(* IEC 61131-3 sources: SRCI/RobotLibrary/Library/POUs/BasicMove/MC_MoveAxesAbsolute, 1 file *)

(* ---- MC_MoveAxesAbsoluteFB.st ---- *)
/// Move all joints to an absolute joint position (Absolute Joint PTP)
FUNCTION_BLOCK MC_MoveAxesAbsoluteFB EXTENDS RobotLibraryBaseExecuteFB
// -------------------------------------------------------------------------
//  SRCI Robot Library
// -------------------------------------------------------------------------
//
//  Object:      MoveAxesAbsoluteFB
//  Author:      Thorsten Brach
//  Date:        2024-06-01
//
//  Description:
//
//
//  Copyright:
//    (C) 2024 Thorsten Brach. All rights reserved
//             Licensed under the LGPL-3.0 license.
//
//  Disclaimer:
//    This project is provided without any guarantee and can be used for
//    private and commercial purposes. Any use is at the user’s
//    own risk and responsibility.
//
// -------------------------------------------------------------------------
VAR_INPUT
  /// Parameter which determines the behavior towards the previously sent and still active or buffered commands
  AbortingMode       : AbortingMode;
  /// Defines the target sequence in which the command will be executed
  SequenceFlag       : SequenceFlag;
  /// command parameter
  ParCmd             : MoveAxesAbsoluteParCmd;
END_VAR

VAR_OUTPUT
  /// Command is transferred and confirmed by the RC
  CommandBuffered    : BOOL;
  /// The command takes control of the motion of the according axis group
  Active             : BOOL;
  /// The command was aborted by another command.
  CommandAborted     : BOOL;
  /// TRUE, while command is interrupted during execution and can be continued
  CommandInterrupted : BOOL;
  /// command results
  OutCmd             : MoveAxesAbsoluteOutCmd;
END_VAR

VAR
  /// internal copy of command parameter
 _parCmd             : MoveAxesAbsoluteParCmd;
  /// command data to send
 _command            : MoveAxesAbsoluteSendData;
  /// response data received
 _response           : MoveAxesAbsoluteRecvData;
END_VAR

  SUPER^(AxesGroup := AxesGroup);

END_FUNCTION_BLOCK

METHOD INTERNAL CheckAddParameter : BOOL
VAR_INPUT
  /// Payload pointer
  PayloadPtr : UDINT;
END_VAR
VAR
  /// Payload as byte array
  Payload    : ARRAY [1..SIZEOF(_command)] OF BYTE;
  /// Null Byte array
  Null       : ARRAY [1..SIZEOF(_command)] OF BYTE;
  /// Data length to compare
  DataLen    : UDINT;
END_VAR

  // Payload pointer must be decreased by one byte, because ADR(Payload) is already one byte !
  PayloadPtr := LIMIT (0, PayloadPtr - 1, SIZEOF(Payload) -1);
  // Convert command struct to payload array
  SysDepMemCpy( pDest := ADR(Payload), pSrc := ADR(_command), DataLen := SIZEOF(_command));
  // Calculate the data length to compare - at least one byte must be compared !
  DataLen := LIMIT(1, SIZEOF(Payload) - PayloadPtr, SIZEOF(Payload));
  // Compare Payload-Array with Null-Byte-Array
  CheckAddParameter := SysDepMemCmp( pData1 := ADR(Payload) + PayloadPtr , pData2 := ADR(Null), DataLen := DataLen) <>  RobotLibraryConstants.OK ;

END_METHOD

METHOD PROTECTED CheckFunctionSupported : BOOL
VAR_IN_OUT
  /// Robot assignment of function
  AxesGroup : AxesGroup;
END_VAR

  CheckFunctionSupported := AxesGroup.State.RobotData.RCSupportedFunctions.MoveAxesAbsolute;

  IF ( NOT CheckFunctionSupported )
  THEN
    // call base implementation for set error and create log entry
    SUPER^.CheckFunctionSupported(AxesGroup := AxesGroup);
  END_IF

END_METHOD

METHOD PROTECTED CheckParameterChanged : BOOL
VAR_IN_OUT
  /// Robot assignment of function
  AxesGroup    : AxesGroup;
END_VAR

  // Check ParCmd Size is > 0, because MemCmp does not work correctly with size = 0
  IF (SIZEOF(ParCmd) = 0) OR (_stepCmd = 0)
  THEN
    RETURN;
  END_IF

  // compare memory
  _parameterChanged := ( SysDepMemCmp(pData1 := ADR(ParCmd), pData2 := ADR(_parCmd), DataLen := SIZEOF(ParCmd)) <> RobotLibraryConstants.OK );

  // check parameter valid ?
  _parameterValid   := CheckParameterValid( AxesGroup := AxesGroup );

  IF ((  _parameterChanged        )  AND
      (  _parameterValid          )) OR
      (  _parameterUpdateInternal )
  THEN
    // reset internal flag for send parameter update
   _parameterUpdateInternal := FALSE;
    // update internal copy of parameters
   _parCmd := ParCmd;
    // inc parameter sequence
   _command.ParSeq := _command.ParSeq + 1;
    // update command data
    CommandData := CreateCommandPayload(AxesGroup := AxesGroup); // ( Access via reference to rCommandFB in ACR )
    // notify active command register
    AxesGroup.Acyclic.ActiveCommandRegister.NotifyParameterChanged := _uniqueID;
  END_IF

END_METHOD

METHOD PROTECTED CheckParameterValid : BOOL
VAR_IN_OUT
  /// Robot assignment of function
  AxesGroup : AxesGroup;
END_VAR
VAR
  /// internal index for loops
 _idx : DINT;
END_VAR

  CheckParameterValid := TRUE;

  // Check AbortingMode valid ?
  IF (( AbortingMode <> AbortingModeEnum.BUFFER ) AND
      ( AbortingMode <> AbortingModeEnum.ABORT  ))
  THEN
    // Parameter not valid
    CheckParameterValid := FALSE;
    // Set error
    ErrorID := RobotLibraryErrorIdEnum.ERR_ABORTINGMODE_INVALID;
    // Create log entry
    CreateLogMessagePara1 ( Timestamp   := AxesGroup.State.SystemTime,
                            MessageType := MessageType.CMD,
                            Severity    := Severity.ERROR,
                            MessageCode := ErrorID,
                            MessageText := 'Invalid Parameter AbortingMode = {1}',
                            Para1       := ABORTING_MODE_TO_STRING(AbortingMode));
    RETURN;
  END_IF

  // Check SequenceFlag valid ?
  IF (( SequenceFlag <> SequenceFlagEnum.PRIMARY_SEQUENCE   ) AND
      ( SequenceFlag <> SequenceFlagEnum.SECONDARY_SEQUENCE ))
  THEN
    // Parameter not valid
    CheckParameterValid := FALSE;
    // Set error
    ErrorID := RobotLibraryErrorIdEnum.ERR_SEQFLAG_NOT_ALLOWED;
    // Create log entry
    CreateLogMessagePara1 ( Timestamp   := AxesGroup.State.SystemTime,
                            MessageType := MessageType.CMD,
                            Severity    := Severity.ERROR,
                            MessageCode := ErrorID,
                            MessageText := 'Invalid Parameter SequenceFlag = {1}',
                            Para1       := SEQUENCE_FLAG_TO_STRING(SequenceFlag));
    RETURN;
  END_IF

  // Check ParCmd.JointPosition.J1 valid ?
  IF ( SysDepIsValidReal(ParCmd.JointPosition.J1) = FALSE )
  THEN
    // Parameter not valid
    CheckParameterValid := FALSE;
    // Set error
    ErrorID := RobotLibraryErrorIdEnum.ERR_INVALID_PAR_CMD;

    // Create log entry
    CreateLogMessagePara1 ( Timestamp   := AxesGroup.State.SystemTime,
                            MessageType := MessageType.CMD,
                            Severity    := Severity.ERROR,
                            MessageCode := ErrorID,
                            MessageText := 'Invalid Parameter ParCmd.JointPosition.J1 = {1}',
                            Para1       := VALID_REAL_TO_STRING(ParCmd.JointPosition.J1));
    RETURN;
  END_IF

  // Check ParCmd.JointPosition.J2 valid ?
  IF ( SysDepIsValidReal(ParCmd.JointPosition.J2) = FALSE )
  THEN
    // Parameter not valid
    CheckParameterValid := FALSE;
    // Set error
    ErrorID := RobotLibraryErrorIdEnum.ERR_INVALID_PAR_CMD;

    // Create log entry
    CreateLogMessagePara1 ( Timestamp   := AxesGroup.State.SystemTime,
                            MessageType := MessageType.CMD,
                            Severity    := Severity.ERROR,
                            MessageCode := ErrorID,
                            MessageText := 'Invalid Parameter ParCmd.JointPosition.J2 = {1}',
                            Para1       := VALID_REAL_TO_STRING(ParCmd.JointPosition.J2));
    RETURN;
  END_IF

  // Check ParCmd.JointPosition.J3 valid ?
  IF ( SysDepIsValidReal(ParCmd.JointPosition.J3) = FALSE )
  THEN
    // Parameter not valid
    CheckParameterValid := FALSE;
    // Set error
    ErrorID := RobotLibraryErrorIdEnum.ERR_INVALID_PAR_CMD;

    // Create log entry
    CreateLogMessagePara1 ( Timestamp   := AxesGroup.State.SystemTime,
                            MessageType := MessageType.CMD,
                            Severity    := Severity.ERROR,
                            MessageCode := ErrorID,
                            MessageText := 'Invalid Parameter ParCmd.JointPosition.J3 = {1}',
                            Para1       := VALID_REAL_TO_STRING(ParCmd.JointPosition.J3));
    RETURN;
  END_IF

  // Check ParCmd.JointPosition.J4 valid ?
  IF ( SysDepIsValidReal(ParCmd.JointPosition.J4) = FALSE )
  THEN
    // Parameter not valid
    CheckParameterValid := FALSE;
    // Set error
    ErrorID := RobotLibraryErrorIdEnum.ERR_INVALID_PAR_CMD;

    // Create log entry
    CreateLogMessagePara1 ( Timestamp   := AxesGroup.State.SystemTime,
                            MessageType := MessageType.CMD,
                            Severity    := Severity.ERROR,
                            MessageCode := ErrorID,
                            MessageText := 'Invalid Parameter ParCmd.JointPosition.J4 = {1}',
                            Para1       := VALID_REAL_TO_STRING(ParCmd.JointPosition.J4));
    RETURN;
  END_IF

  // Check ParCmd.JointPosition.J5 valid ?
  IF ( SysDepIsValidReal(ParCmd.JointPosition.J5) = FALSE )
  THEN
    // Parameter not valid
    CheckParameterValid := FALSE;
    // Set error
    ErrorID := RobotLibraryErrorIdEnum.ERR_INVALID_PAR_CMD;

    // Create log entry
    CreateLogMessagePara1 ( Timestamp   := AxesGroup.State.SystemTime,
                            MessageType := MessageType.CMD,
                            Severity    := Severity.ERROR,
                            MessageCode := ErrorID,
                            MessageText := 'Invalid Parameter ParCmd.JointPosition.J5 = {1}',
                            Para1       := VALID_REAL_TO_STRING(ParCmd.JointPosition.J5));
    RETURN;
  END_IF

  // Check ParCmd.JointPosition.J6 valid ?
  IF ( SysDepIsValidReal(ParCmd.JointPosition.J6) = FALSE )
  THEN
    // Parameter not valid
    CheckParameterValid := FALSE;
    // Set error
    ErrorID := RobotLibraryErrorIdEnum.ERR_INVALID_PAR_CMD;

    // Create log entry
    CreateLogMessagePara1 ( Timestamp   := AxesGroup.State.SystemTime,
                            MessageType := MessageType.CMD,
                            Severity    := Severity.ERROR,
                            MessageCode := ErrorID,
                            MessageText := 'Invalid Parameter ParCmd.JointPosition.J6 = {1}',
                            Para1       := VALID_REAL_TO_STRING(ParCmd.JointPosition.J6));
    RETURN;
  END_IF

  // Check ParCmd.JointPosition.E1 valid ?
  IF ( SysDepIsValidReal(ParCmd.JointPosition.E1) = FALSE )
  THEN
    // Parameter not valid
    CheckParameterValid := FALSE;
    // Set error
    ErrorID := RobotLibraryErrorIdEnum.ERR_INVALID_PAR_CMD;

    // Create log entry
    CreateLogMessagePara1 ( Timestamp   := AxesGroup.State.SystemTime,
                            MessageType := MessageType.CMD,
                            Severity    := Severity.ERROR,
                            MessageCode := ErrorID,
                            MessageText := 'Invalid Parameter ParCmd.JointPosition.E1 = {1}',
                            Para1       := VALID_REAL_TO_STRING(ParCmd.JointPosition.E1));
    RETURN;
  END_IF

  // Check ParCmd.JointPosition.E2 valid ?
  IF ( SysDepIsValidReal(ParCmd.JointPosition.E2) = FALSE )
  THEN
    // Parameter not valid
    CheckParameterValid := FALSE;
    // Set error
    ErrorID := RobotLibraryErrorIdEnum.ERR_INVALID_PAR_CMD;

    // Create log entry
    CreateLogMessagePara1 ( Timestamp   := AxesGroup.State.SystemTime,
                            MessageType := MessageType.CMD,
                            Severity    := Severity.ERROR,
                            MessageCode := ErrorID,
                            MessageText := 'Invalid Parameter ParCmd.JointPosition.E2 = {1}',
                            Para1       := VALID_REAL_TO_STRING(ParCmd.JointPosition.E2));
    RETURN;
  END_IF

  // Check ParCmd.JointPosition.E3 valid ?
  IF ( SysDepIsValidReal(ParCmd.JointPosition.E3) = FALSE )
  THEN
    // Parameter not valid
    CheckParameterValid := FALSE;
    // Set error
    ErrorID := RobotLibraryErrorIdEnum.ERR_INVALID_PAR_CMD;

    // Create log entry
    CreateLogMessagePara1 ( Timestamp   := AxesGroup.State.SystemTime,
                            MessageType := MessageType.CMD,
                            Severity    := Severity.ERROR,
                            MessageCode := ErrorID,
                            MessageText := 'Invalid Parameter ParCmd.JointPosition.E3 = {1}',
                            Para1       := VALID_REAL_TO_STRING(ParCmd.JointPosition.E3));
    RETURN;
  END_IF

  // Check ParCmd.JointPosition.E4 valid ?
  IF ( SysDepIsValidReal(ParCmd.JointPosition.E4) = FALSE )
  THEN
    // Parameter not valid
    CheckParameterValid := FALSE;
    // Set error
    ErrorID := RobotLibraryErrorIdEnum.ERR_INVALID_PAR_CMD;

    // Create log entry
    CreateLogMessagePara1 ( Timestamp   := AxesGroup.State.SystemTime,
                            MessageType := MessageType.CMD,
                            Severity    := Severity.ERROR,
                            MessageCode := ErrorID,
                            MessageText := 'Invalid Parameter ParCmd.JointPosition.E4 = {1}',
                            Para1       := VALID_REAL_TO_STRING(ParCmd.JointPosition.E4));
    RETURN;
  END_IF

  // Check ParCmd.JointPosition.E5 valid ?
  IF ( SysDepIsValidReal(ParCmd.JointPosition.E5) = FALSE )
  THEN
    // Parameter not valid
    CheckParameterValid := FALSE;
    // Set error
    ErrorID := RobotLibraryErrorIdEnum.ERR_INVALID_PAR_CMD;

    // Create log entry
    CreateLogMessagePara1 ( Timestamp   := AxesGroup.State.SystemTime,
                            MessageType := MessageType.CMD,
                            Severity    := Severity.ERROR,
                            MessageCode := ErrorID,
                            MessageText := 'Invalid Parameter ParCmd.JointPosition.E5 = {1}',
                            Para1       := VALID_REAL_TO_STRING(ParCmd.JointPosition.E5));
    RETURN;
  END_IF

  // Check ParCmd.JointPosition.E6 valid ?
  IF ( SysDepIsValidReal(ParCmd.JointPosition.E6) = FALSE )
  THEN
    // Parameter not valid
    CheckParameterValid := FALSE;
    // Set error
    ErrorID := RobotLibraryErrorIdEnum.ERR_INVALID_PAR_CMD;

    // Create log entry
    CreateLogMessagePara1 ( Timestamp   := AxesGroup.State.SystemTime,
                            MessageType := MessageType.CMD,
                            Severity    := Severity.ERROR,
                            MessageCode := ErrorID,
                            MessageText := 'Invalid Parameter ParCmd.JointPosition.E6 = {1}',
                            Para1       := VALID_REAL_TO_STRING(ParCmd.JointPosition.E6));
    RETURN;
  END_IF

  // Check ParCmd.VelocityRate valid ?
  IF  (( SysDepIsValidReal(ParCmd.VelocityRate) = FALSE )  OR
      ((                   ParCmd.VelocityRate  <     0 )  AND
       (                   ParCmd.VelocityRate <>    -1 )) OR
       (                   ParCmd.VelocityRate  >   100 ))
  THEN
    // Parameter not valid
    CheckParameterValid := FALSE;
    // Set error
    ErrorID := RobotLibraryErrorIdEnum.ERR_VELOCITY_INVALID;
    // Create log entry
    CreateLogMessagePara1 ( Timestamp   := AxesGroup.State.SystemTime,
                            MessageType := MessageType.CMD,
                            Severity    := Severity.ERROR,
                            MessageCode := ErrorID,
                            MessageText := 'Invalid Parameter ParCmd.VelocityRate = {1}',
                            Para1       := VALID_REAL_TO_STRING(ParCmd.VelocityRate));
    RETURN;
  END_IF

  // Check ParCmd.AccelerationRate valid ?
  IF  (( SysDepIsValidReal(ParCmd.AccelerationRate) = FALSE )  OR
      ((                   ParCmd.AccelerationRate  <     0 )  AND
       (                   ParCmd.AccelerationRate <>    -1 )) OR
       (                   ParCmd.AccelerationRate  >   100 ))
  THEN
    // Parameter not valid
    CheckParameterValid := FALSE;
    // Set error
    ErrorID := RobotLibraryErrorIdEnum.ERR_ACCELERATION_INVALID;
    // Create log entry
    CreateLogMessagePara1 ( Timestamp   := AxesGroup.State.SystemTime,
                            MessageType := MessageType.CMD,
                            Severity    := Severity.ERROR,
                            MessageCode := ErrorID,
                            MessageText := 'Invalid Parameter ParCmd.AccelerationRate = {1}',
                            Para1       := VALID_REAL_TO_STRING(ParCmd.AccelerationRate));
    RETURN;
  END_IF

  // Check ParCmd.DecelerationRate valid ?
  IF  (( SysDepIsValidReal(ParCmd.DecelerationRate) = FALSE )  OR
      ((                   ParCmd.DecelerationRate  <     0 )  AND
       (                   ParCmd.DecelerationRate <>    -1 )) OR
       (                   ParCmd.DecelerationRate  >   100 ))
  THEN
    // Parameter not valid
    CheckParameterValid := FALSE;
    // Set error
    ErrorID := RobotLibraryErrorIdEnum.ERR_DECELERATION_INVALID;
    // Create log entry
    CreateLogMessagePara1 ( Timestamp   := AxesGroup.State.SystemTime,
                            MessageType := MessageType.CMD,
                            Severity    := Severity.ERROR,
                            MessageCode := ErrorID,
                            MessageText := 'Invalid Parameter ParCmd.DecelerationRate = {1}',
                            Para1       := VALID_REAL_TO_STRING(ParCmd.DecelerationRate));
    RETURN;
  END_IF

  // Check ParCmd.JerkRate valid ?
  IF  (( SysDepIsValidReal(ParCmd.JerkRate) = FALSE )  OR
      ((                   ParCmd.JerkRate  <     0 )  AND
       (                   ParCmd.JerkRate <>    -1 )) OR
       (                   ParCmd.JerkRate  >   100 ))
  THEN
    // Parameter not valid
    CheckParameterValid := FALSE;
    // Set error
    ErrorID := RobotLibraryErrorIdEnum.ERR_JERK_INVALID;
    // Create log entry
    CreateLogMessagePara1 ( Timestamp   := AxesGroup.State.SystemTime,
                            MessageType := MessageType.CMD,
                            Severity    := Severity.ERROR,
                            MessageCode := ErrorID,
                            MessageText := 'Invalid Parameter ParCmd.JerkRate = {1}',
                            Para1       := VALID_REAL_TO_STRING(ParCmd.JerkRate));
    RETURN;
  END_IF

  // Check ParCmd.ToolNo valid ?
  IF (( ParCmd.ToolNo <   0                                                ) OR
      ( ParCmd.ToolNo > 254                                                ) OR
      ( ParCmd.ToolNo > AxesGroup.State.ConfigurationData.HighestToolIndex ) OR
      ( ParCmd.ToolNo > RobotLibraryParameter.TOOL_MAX -1                  ))
  THEN
    // Parameter not valid
    CheckParameterValid := FALSE;

    // Check ToolNo available on RC ?
    IF ( ParCmd.ToolNo > AxesGroup.State.ConfigurationData.HighestToolIndex )
    THEN
      ErrorID := RobotLibraryErrorIdEnum.ERR_TOOLNO_UNAVAILABLE;
    ELSE
      ErrorID := RobotLibraryErrorIdEnum.ERR_TOOLNO_RANGE;
  	END_IF

    // Create log entry
    CreateLogMessagePara1 ( Timestamp   := AxesGroup.State.SystemTime,
                            MessageType := MessageType.CMD,
                            Severity    := Severity.ERROR,
                            MessageCode := ErrorID,
                            MessageText := 'Invalid Parameter ParCmd.ToolNo = {1}',
                            Para1       := USINT_TO_STRING(ParCmd.ToolNo));
    RETURN;
  END_IF

  // Check ParCmd.BlendingMode valid ?
  IF (( ParCmd.BlendingMode <> BlendingMode.EXACT_STOP           ) AND
      ( ParCmd.BlendingMode <> BlendingMode.DEFINED_VELOCITY     ) AND
      ( ParCmd.BlendingMode <> BlendingMode.CORNER_DISTANCE      ) AND
      ( ParCmd.BlendingMode <> BlendingMode.MAX_CORNER_DEVIATION ) AND
      ( ParCmd.BlendingMode <> BlendingMode.CORNER_DISTANCE_2R   ) AND
      ( ParCmd.BlendingMode <> BlendingMode.RAMP_OVERLAP         ) AND
      ( ParCmd.BlendingMode <> BlendingMode.CORNER_DISTANCE_1R   ))
  THEN
    // Parameter not valid
    CheckParameterValid := FALSE;
    // Set error
    ErrorID := RobotLibraryErrorIdEnum.ERR_INVALID_PAR_CMD;
    // Create log entry
    CreateLogMessagePara1 ( Timestamp   := AxesGroup.State.SystemTime,
                            MessageType := MessageType.CMD,
                            Severity    := Severity.ERROR,
                            MessageCode := ErrorID,
                            MessageText := 'Invalid Parameter ParCmd.BlendingMode = {1}',
                            Para1       := BLENDING_MODE_TO_STRING(ParCmd.BlendingMode));
    RETURN;
  END_IF

  FOR _idx := 0 TO 1
  DO
    // Check ParCmd.BlendingParameter valid ?
    IF  ( SysDepIsValidReal(ParCmd.BlendingParameter[_idx]) = FALSE )
    THEN
      // Parameter not valid
      CheckParameterValid := FALSE;
      // Set error
      ErrorID := RobotLibraryErrorIdEnum.ERR_JERK_INVALID;
      // Create log entry
      CreateLogMessagePara2 ( Timestamp   := AxesGroup.State.SystemTime,
                              MessageType := MessageType.CMD,
                              Severity    := Severity.ERROR,
                              MessageCode := ErrorID,
                              MessageText := 'Invalid Parameter ParCmd.BlendingParameter[{2}] = {1}',
                              Para1       := VALID_REAL_TO_STRING(ParCmd.JerkRate),
                              Para2       := DINT_TO_STRING(_idx));
      EXIT;
      RETURN;
    END_IF
  END_FOR

  // Check ParCmd.MoveTime valid ?
  IF  ( ParCmd.MoveTime < T#0S )
  THEN
    // Parameter not valid
    CheckParameterValid := FALSE;
    // Set error
    ErrorID := RobotLibraryErrorIdEnum.ERR_INVALID_PAR_CMD;
    // Create log entry
    CreateLogMessagePara1 ( Timestamp   := AxesGroup.State.SystemTime,
                            MessageType := MessageType.CMD,
                            Severity    := Severity.ERROR,
                            MessageCode := ErrorID,
                            MessageText := 'Invalid Parameter ParCmd.MoveTime = {1}',
                            Para1       := TIME_TO_STRING(ParCmd.MoveTime));
    RETURN;
  END_IF

  // Check ParCmd.Manipulation
  // -> no plausibility check for boolean

  FOR _idx := 0 TO 3
  DO
    // Check ParCmd.EmitterID valid ?
    IF  (( ParCmd.EmitterID[_idx] < -127 ) OR
         ( ParCmd.EmitterID[_idx] >  127 ))
    THEN
      // Parameter not valid
      CheckParameterValid := FALSE;
      // Set error
      ErrorID := RobotLibraryErrorIdEnum.ERR_INVALID_PAR_CMD;
      // Create log entry
      CreateLogMessagePara2 ( Timestamp   := AxesGroup.State.SystemTime,
                              MessageType := MessageType.CMD,
                              Severity    := Severity.ERROR,
                              MessageCode := ErrorID,
                              MessageText := 'Invalid Parameter ParCmd.EmitterID[{2}] = {1}',
                              Para1       := SINT_TO_STRING(ParCmd.EmitterID[_idx]),
                              Para2       := DINT_TO_STRING(_idx));
      EXIT;
      RETURN;
    END_IF
  END_FOR

END_METHOD

METHOD INTERNAL CreateCommandPayload : RobotLibraryCommandDataFB
VAR_IN_OUT
  /// Robot assignment of function
  AxesGroup : AxesGroup;
END_VAR
VAR
  /// internal index for loops
 _idx          : DINT;
  /// Parameter count
 _parameterCnt : DINT;
END_VAR
// Table 6-261: Sent CMD payload (PLC to RC) of "MoveAxesAbsolute
// --------------------------
// Header
// --------------------------
// --------------------------
// Datablock
// --------------------------
// Byte 00 : UINT  - Type HB
// Byte 01 :       - Type LB
// Byte 02 : USINT - Reserve | ExecutionMode
// Byte 03 : USINT - ParSeq  | Priority
// --------------------------
// Datablock
// --------------------------
// Byte 04 : SINT       - EmitterID[0]
// Byte 05 : SINT       - EmitterID[1]
// Byte 06 : SINT       - EmitterID[2]
// Byte 07 : SINT       - EmitterID[3]
// Byte 08 : SINT       - ListenerID
// Byte 09 : BYTE       - Reserved
// Byte 10 : UINT       - VelocityRate HW HB
// Byte 11 :            - VelocityRate HW LB
// Byte 12 : UINT       - AccelerationRate HW HB
// Byte 13 :            - AccelerationRate HW LB
// Byte 14 : UINT       - DecelerationRate HW HB
// Byte 15 :            - DecelerationRate HW LB
// Byte 16 : UINT       - JerkRate HW HB
// Byte 17 :            - JerkRate HW LB
// Byte 18 : USINT      - ToolNo
// Byte 19 : USINT      - BlendingMode
// Byte 20 : REAL       - BlendingParameter[0] HW HB
// Byte 21 :            - BlendingParameter[0] HW LB
// Byte 22 :            - BlendingParameter[0] LW HB
// Byte 23 :            - BlendingParameter[0] LW LB
// Byte 24 : REAL       - BlendingParameter[1] HW HB
// Byte 25 :            - BlendingParameter[1] HW LB
// Byte 26 :            - BlendingParameter[1] LW HB
// Byte 27 :            - BlendingParameter[1] LW LB
// Byte 28 : REAL       - JointPosition.J1 HW HB
// Byte 29 :            - JointPosition.J1 HW LB
// Byte 30 :            - JointPosition.J1 LW HB
// Byte 31 :            - JointPosition.J1 LW LB
// Byte 32 : REAL       - JointPosition.J2 HW HB
// Byte 33 :            - JointPosition.J2 HW LB
// Byte 34 :            - JointPosition.J2 LW HB
// Byte 35 :            - JointPosition.J2 LW LB
// Byte 36 : REAL       - JointPosition.J3 HW HB
// Byte 37 :            - JointPosition.J3 HW LB
// Byte 38 :            - JointPosition.J3 LW HB
// Byte 39 :            - JointPosition.J3 LW LB
// Byte 40 : REAL       - JointPosition.J4 HW HB
// Byte 41 :            - JointPosition.J4 HW LB
// Byte 42 :            - JointPosition.J4 LW HB
// Byte 43 :            - JointPosition.J4 LW LB
// Byte 44 : REAL       - JointPosition.J5 HW HB
// Byte 45 :            - JointPosition.J5 HW LB
// Byte 46 :            - JointPosition.J5 LW HB
// Byte 47 :            - JointPosition.J5 LW LB
// Byte 48 : REAL       - JointPosition.J6 HW HB
// Byte 49 :            - JointPosition.J6 HW LB
// Byte 50 :            - JointPosition.J6 LW HB
// Byte 51 :            - JointPosition.J6 LW LB
// Byte 52 : REAL       - JointPosition.E1 HW HB
// Byte 53 :            - JointPosition.E1 HW LB
// Byte 54 :            - JointPosition.E1 LW HB
// Byte 55 :            - JointPosition.E1 LW LB
// Byte 56 : BOOL       - Manipulation
// Byte 57 : BYTE       - Reserve
// Byte 58 : UINT       - Time HW HB
// Byte 59 :            - Time HW LB
// Byte 60 : REAL       - JointPosition.E2 HW HB
// Byte 61 :            - JointPosition.E2 HW LB
// Byte 62 :            - JointPosition.E2 LW HB
// Byte 63 :            - JointPosition.E2 LW LB
// Byte 64 : REAL       - JointPosition.E3 HW HB
// Byte 65 :            - JointPosition.E3 HW LB
// Byte 66 :            - JointPosition.E3 LW HB
// Byte 67 :            - JointPosition.E3 LW LB
// Byte 68 : REAL       - JointPosition.E4 HW HB
// Byte 69 :            - JointPosition.E4 HW LB
// Byte 70 :            - JointPosition.E4 LW HB
// Byte 71 :            - JointPosition.E4 LW LB
// Byte 72 : REAL       - JointPosition.E5 HW HB
// Byte 73 :            - JointPosition.E5 HW LB
// Byte 74 :            - JointPosition.E5 LW HB
// Byte 75 :            - JointPosition.E5 LW LB
// Byte 76 : REAL       - JointPosition.E6 HW HB
// Byte 77 :            - JointPosition.E6 HW LB
// Byte 78 :            - JointPosition.E6 LW HB
// Byte 79 :            - JointPosition.E6 LW LB

  // set command parameter
  _command.CmdTyp            :=  CmdType.MoveAxesAbsolute;
  _command.ExecMode          :=  ExecMode;
  _command.ParSeq            := _command.ParSeq;
  _command.Priority          :=  Priority;
  _command.EmitterID[0]      := _parCmd.EmitterID[0];
  _command.EmitterID[1]      := _parCmd.EmitterID[1];
  _command.EmitterID[2]      := _parCmd.EmitterID[2];
  _command.EmitterID[3]      := _parCmd.EmitterID[3];
  _command.ListenerID        := 0;
  _command.Reserve           := 0;

  _command.VelocityRate      := REAL_TO_PERCENT_UINT(_parCmd.VelocityRate     , IsOptional := FALSE);
  _command.AccelerationRate  := REAL_TO_PERCENT_UINT(_parCmd.AccelerationRate , IsOptional := FALSE);
  _command.JerkRate          := REAL_TO_PERCENT_UINT(_parCmd.JerkRate         , IsOptional := TRUE );
  _command.DecelerationRate  := REAL_TO_PERCENT_UINT(_parCmd.DecelerationRate , IsOptional := TRUE );

  _command.ToolNo            := _parCmd.ToolNo;
  _command.BlendingMode      := _parCmd.BlendingMode;
  _command.BlendingParameter := _parCmd.BlendingParameter;
  _command.JointPosition     := _parCmd.JointPosition;
  _command.Manipulation      := _parCmd.Manipulation;
  _command.MoveTime          := TIME_TO_UINT(_parCmd.MoveTime);

  // copy command data to header
  _cmdHeader := _command;
  // call base implementation to copy header to payload buffer
  CreateCommandPayload := SUPER^.CreateCommandPayload(AxesGroup := AxesGroup);

  FOR _idx := 0 TO 3
  DO
    // Check parameter must be added ?
    IF ( CheckAddParameter(CreateCommandPayload.PayloadPtr))
    THEN
      // add command.EmitterID[x]
      CreateCommandPayload.AddSint(_command.EmitterID[_idx]);
      // inc parameter counter
     _parameterCnt := _parameterCnt + 1;
    END_IF
  END_FOR

  // Check parameter must be added ?
  IF ( CheckAddParameter(CreateCommandPayload.PayloadPtr))
  THEN
    // add command.ListenerID
    CreateCommandPayload.AddSint(_command.ListenerID);
    // inc parameter counter
   _parameterCnt := _parameterCnt + 1;
  END_IF

  // Check parameter must be added ?
  IF ( CheckAddParameter(CreateCommandPayload.PayloadPtr))
  THEN
    // add command.Reserve
    CreateCommandPayload.AddSint(_command.Reserve);
    // inc parameter counter
   _parameterCnt := _parameterCnt + 1;
  END_IF

  // Check parameter must be added ?
  IF ( CheckAddParameter(CreateCommandPayload.PayloadPtr))
  THEN
    // add command.VelocityRate
    CreateCommandPayload.AddUint(_command.VelocityRate);
    // inc parameter counter
   _parameterCnt := _parameterCnt + 1;
  END_IF

  // Check parameter must be added ?
  IF ( CheckAddParameter(CreateCommandPayload.PayloadPtr))
  THEN
    // add command.AccelerationRate
    CreateCommandPayload.AddUint(_command.AccelerationRate);
    // inc parameter counter
   _parameterCnt := _parameterCnt + 1;
  END_IF

  // Check parameter must be added ?
  IF ( CheckAddParameter(CreateCommandPayload.PayloadPtr))
  THEN
    // add command.DecelerationRate
    CreateCommandPayload.AddUint(_command.DecelerationRate);
    // inc parameter counter
   _parameterCnt := _parameterCnt + 1;
  END_IF

  // Check parameter must be added ?
  IF ( CheckAddParameter(CreateCommandPayload.PayloadPtr))
  THEN
    // add command.JerkRate
    CreateCommandPayload.AddUint(_command.JerkRate);
    // inc parameter counter
   _parameterCnt := _parameterCnt + 1;
  END_IF

  // Check parameter must be added ?
  IF ( CheckAddParameter(CreateCommandPayload.PayloadPtr))
  THEN
    // add command.ToolNo
    CreateCommandPayload.AddUsint(_command.ToolNo);
    // inc parameter counter
   _parameterCnt := _parameterCnt + 1;
  END_IF

  // Check parameter must be added ?
  IF ( CheckAddParameter(CreateCommandPayload.PayloadPtr))
  THEN
    // add command.BlendingMode
    CreateCommandPayload.AddUsint(_command.BlendingMode);
    // inc parameter counter
   _parameterCnt := _parameterCnt + 1;
  END_IF

  // Check parameter must be added ?
  IF ( CheckAddParameter(CreateCommandPayload.PayloadPtr))
  THEN
    // add command.BlendingParameter[0]
    CreateCommandPayload.AddReal(_command.BlendingParameter[0]);
    // inc parameter counter
   _parameterCnt := _parameterCnt + 1;
  END_IF

  // Check parameter must be added ?
  IF ( CheckAddParameter(CreateCommandPayload.PayloadPtr))
  THEN
    // add command.BlendingParameter[1]
    CreateCommandPayload.AddReal(_command.BlendingParameter[1]);
    // inc parameter counter
   _parameterCnt := _parameterCnt + 1;
  END_IF

  // Check parameter must be added ?
  IF ( CheckAddParameter(CreateCommandPayload.PayloadPtr))
  THEN
    // add command.JointPosition.J1
    CreateCommandPayload.AddReal(_command.JointPosition.J1);
    // inc parameter counter
   _parameterCnt := _parameterCnt + 1;
  END_IF

  // Check parameter must be added ?
  IF ( CheckAddParameter(CreateCommandPayload.PayloadPtr))
  THEN
    // add command.JointPosition.J2
    CreateCommandPayload.AddReal(_command.JointPosition.J2);
    // inc parameter counter
   _parameterCnt := _parameterCnt + 1;
  END_IF

  // Check parameter must be added ?
  IF ( CheckAddParameter(CreateCommandPayload.PayloadPtr))
  THEN
    // add command.JointPosition.J3
    CreateCommandPayload.AddReal(_command.JointPosition.J3);
    // inc parameter counter
   _parameterCnt := _parameterCnt + 1;
  END_IF

  // Check parameter must be added ?
  IF ( CheckAddParameter(CreateCommandPayload.PayloadPtr))
  THEN
    // add command.JointPosition.J4
    CreateCommandPayload.AddReal(_command.JointPosition.J4);
    // inc parameter counter
   _parameterCnt := _parameterCnt + 1;
  END_IF

  // Check parameter must be added ?
  IF ( CheckAddParameter(CreateCommandPayload.PayloadPtr))
  THEN
    // add command.JointPosition.J5
    CreateCommandPayload.AddReal(_command.JointPosition.J5);
    // inc parameter counter
   _parameterCnt := _parameterCnt + 1;
  END_IF

  // Check parameter must be added ?
  IF ( CheckAddParameter(CreateCommandPayload.PayloadPtr))
  THEN
    // add command.JointPosition.J6
    CreateCommandPayload.AddReal(_command.JointPosition.J6);
    // inc parameter counter
   _parameterCnt := _parameterCnt + 1;
  END_IF

  // Check parameter must be added ?
  IF ( CheckAddParameter(CreateCommandPayload.PayloadPtr))
  THEN
    // add command.JointPosition.E1
    CreateCommandPayload.AddReal(_command.JointPosition.E1);
    // inc parameter counter
   _parameterCnt := _parameterCnt + 1;
  END_IF

  // Check parameter must be added ?
  IF ( CheckAddParameter(CreateCommandPayload.PayloadPtr))
  THEN
    // add command.Manipulation
    CreateCommandPayload.AddBool(_command.Manipulation);
    // inc parameter counter
   _parameterCnt := _parameterCnt + 1;
  END_IF

  // Check parameter must be added ?
  IF ( CheckAddParameter(CreateCommandPayload.PayloadPtr))
  THEN
    // add command.Reserve
    CreateCommandPayload.AddByte(_command.Reserve2);
    // inc parameter counter
   _parameterCnt := _parameterCnt + 1;
  END_IF

  // Check parameter must be added ?
  IF ( CheckAddParameter(CreateCommandPayload.PayloadPtr))
  THEN
    // add command.MoveTime
    CreateCommandPayload.AddUint(_command.MoveTime);
    // inc parameter counter
   _parameterCnt := _parameterCnt + 1;
  END_IF

  // Check parameter must be added ?
  IF ( CheckAddParameter(CreateCommandPayload.PayloadPtr))
  THEN
    // add command.JointPosition.E2
    CreateCommandPayload.AddReal(_command.JointPosition.E2);
    // inc parameter counter
   _parameterCnt := _parameterCnt + 1;
  END_IF

  // Check parameter must be added ?
  IF ( CheckAddParameter(CreateCommandPayload.PayloadPtr))
  THEN
    // add command.JointPosition.E3
    CreateCommandPayload.AddReal(_command.JointPosition.E3);
    // inc parameter counter
   _parameterCnt := _parameterCnt + 1;
  END_IF

  // Check parameter must be added ?
  IF ( CheckAddParameter(CreateCommandPayload.PayloadPtr))
  THEN
    // add command.JointPosition.E4
    CreateCommandPayload.AddReal(_command.JointPosition.E4);
    // inc parameter counter
   _parameterCnt := _parameterCnt + 1;
  END_IF

  // Check parameter must be added ?
  IF ( CheckAddParameter(CreateCommandPayload.PayloadPtr))
  THEN
    // add command.JointPosition.E5
    CreateCommandPayload.AddReal(_command.JointPosition.E5);
    // inc parameter counter
   _parameterCnt := _parameterCnt + 1;
  END_IF

  // Check parameter must be added ?
  IF ( CheckAddParameter(CreateCommandPayload.PayloadPtr))
  THEN
    // add command.JointPosition.E6
    CreateCommandPayload.AddReal(_command.JointPosition.E6);
    // inc parameter counter
   _parameterCnt := _parameterCnt + 1;
  END_IF

  // create logging
  CreateCommandPayloadLog(AxesGroup := AxesGroup, ParameterCnt := _parameterCnt);

END_METHOD

METHOD INTERNAL CreateCommandPayloadLog
VAR_IN_OUT
  /// Robot assignment of function
  AxesGroup : AxesGroup;
END_VAR
VAR_INPUT
  /// Parameter count
  ParameterCnt : DINT;
END_VAR
VAR
  /// internal index for loops
 _idx : DINT;
END_VAR

  // Create log entry for Parameter start
  CreateLogMessagePara1 ( Timestamp   := AxesGroup.State.SystemTime,
                          MessageType := MessageType.CMD,
                          Severity    := Severity.DEBUG,
                          MessageCode := 0,
                          MessageText := 'Create command payload with the {1} parameter(s) :',
                          Para1       := DINT_TO_STRING(ParameterCnt));

  // Create log entry for EmitterID[x]
  FOR _idx := 0 TO 3
  DO
    // Return if no parameter is remaining...
    IF ( ParameterCnt = 0 ) THEN RETURN; END_IF
    // dec remaining parameter(s)
    ParameterCnt := ParameterCnt - 1;
    // Create log entry for Command.EmitterID
    CreateLogMessagePara2 ( Timestamp   := AxesGroup.State.SystemTime,
                            MessageType := MessageType.CMD,
                            Severity    := Severity.DEBUG,
                            MessageCode := 0,
                            MessageText := 'Command.EmitterID[{2}] = {1}',
                            Para1       :=  SINT_TO_STRING(_command.EmitterID[_idx]),
                            Para2       :=  DINT_TO_STRING(_idx));
  END_FOR

  // Return if no parameter is remaining...
  IF ( ParameterCnt = 0 ) THEN RETURN; END_IF
  // dec remaining parameter(s)
  ParameterCnt := ParameterCnt - 1;
  // Create log entry for ListenerID
  CreateLogMessagePara1 ( Timestamp   := AxesGroup.State.SystemTime,
                          MessageType := MessageType.CMD,
                          Severity    := Severity.DEBUG,
                          MessageCode := 0,
                          MessageText := 'Command.ListenerID = {1}',
                          Para1       :=  SINT_TO_STRING(_command.ListenerID));

  // Return if no parameter is remaining...
  IF ( ParameterCnt = 0 ) THEN RETURN; END_IF
  // dec remaining parameter(s)
  ParameterCnt := ParameterCnt - 1;
  // Create log entry for Reserve
  CreateLogMessagePara1 ( Timestamp   := AxesGroup.State.SystemTime,
                          MessageType := MessageType.CMD,
                          Severity    := Severity.DEBUG,
                          MessageCode := 0,
                          MessageText := 'Command.Reserve = {1}',
                          Para1       :=  SINT_TO_STRING(_command.Reserve));

  // Return if no parameter is remaining...
  IF ( ParameterCnt = 0 ) THEN RETURN; END_IF
  // dec remaining parameter(s)
  ParameterCnt := ParameterCnt - 1;
  // Create log entry for VelocityRate
  CreateLogMessagePara1 ( Timestamp   := AxesGroup.State.SystemTime,
                          MessageType := MessageType.CMD,
                          Severity    := Severity.DEBUG,
                          MessageCode := 0,
                          MessageText := 'Command.VelocityRate = {1}',
                          Para1       :=  UINT_TO_STRING(_command.VelocityRate));

  // Return if no parameter is remaining...
  IF ( ParameterCnt = 0 ) THEN RETURN; END_IF
  // dec remaining parameter(s)
  ParameterCnt := ParameterCnt - 1;
  // Create log entry for AccelerationRate
  CreateLogMessagePara1 ( Timestamp   := AxesGroup.State.SystemTime,
                          MessageType := MessageType.CMD,
                          Severity    := Severity.DEBUG,
                          MessageCode := 0,
                          MessageText := 'Command.AccelerationRate = {1}',
                          Para1       :=  UINT_TO_STRING(_command.AccelerationRate));

  // Return if no parameter is remaining...
  IF ( ParameterCnt = 0 ) THEN RETURN; END_IF
  // dec remaining parameter(s)
  ParameterCnt := ParameterCnt - 1;
  // Create log entry for DecelerationRate
  CreateLogMessagePara1 ( Timestamp   := AxesGroup.State.SystemTime,
                          MessageType := MessageType.CMD,
                          Severity    := Severity.DEBUG,
                          MessageCode := 0,
                          MessageText := 'Command.DecelerationRate = {1}',
                          Para1       :=  UINT_TO_STRING(_command.DecelerationRate));

  // Return if no parameter is remaining...
  IF ( ParameterCnt = 0 ) THEN RETURN; END_IF
  // dec remaining parameter(s)
  ParameterCnt := ParameterCnt - 1;
  // Create log entry for JerkRate
  CreateLogMessagePara1 ( Timestamp   := AxesGroup.State.SystemTime,
                          MessageType := MessageType.CMD,
                          Severity    := Severity.DEBUG,
                          MessageCode := 0,
                          MessageText := 'Command.JerkRate = {1}',
                          Para1       :=  UINT_TO_STRING(_command.JerkRate));

  // Return if no parameter is remaining...
  IF ( ParameterCnt = 0 ) THEN RETURN; END_IF
  // dec remaining parameter(s)
  ParameterCnt := ParameterCnt - 1;
  // Create log entry for ToolNo
  CreateLogMessagePara1 ( Timestamp   := AxesGroup.State.SystemTime,
                          MessageType := MessageType.CMD,
                          Severity    := Severity.DEBUG,
                          MessageCode := 0,
                          MessageText := 'Command.ToolNo = {1}',
                          Para1       :=  USINT_TO_STRING(_command.ToolNo));

  // Return if no parameter is remaining...
  IF ( ParameterCnt = 0 ) THEN RETURN; END_IF
  // dec remaining parameter(s)
  ParameterCnt := ParameterCnt - 1;
  // Create log entry for BlendingMode
  CreateLogMessagePara1 ( Timestamp   := AxesGroup.State.SystemTime,
                          MessageType := MessageType.CMD,
                          Severity    := Severity.DEBUG,
                          MessageCode := 0,
                          MessageText := 'Command.BlendingMode = {1}',
                          Para1       :=  BLENDING_MODE_TO_STRING(_command.BlendingMode));

  // Return if no parameter is remaining...
  IF ( ParameterCnt = 0 ) THEN RETURN; END_IF
  // dec remaining parameter(s)
  ParameterCnt := ParameterCnt - 1;
  // Create log entry for BlendingParameter[0]
  CreateLogMessagePara1 ( Timestamp   := AxesGroup.State.SystemTime,
                          MessageType := MessageType.CMD,
                          Severity    := Severity.DEBUG,
                          MessageCode := 0,
                          MessageText := 'Command.BlendingParameter[0] = {1}',
                          Para1       :=  REAL_TO_STRING(_command.BlendingParameter[0]));

  // Return if no parameter is remaining...
  IF ( ParameterCnt = 0 ) THEN RETURN; END_IF
  // dec remaining parameter(s)
  ParameterCnt := ParameterCnt - 1;
  // Create log entry for BlendingParameter[1]
  CreateLogMessagePara1 ( Timestamp   := AxesGroup.State.SystemTime,
                          MessageType := MessageType.CMD,
                          Severity    := Severity.DEBUG,
                          MessageCode := 0,
                          MessageText := 'Command.BlendingParameter[1] = {1}',
                          Para1       :=  REAL_TO_STRING(_command.BlendingParameter[1]));

  // Return if no parameter is remaining...
  IF ( ParameterCnt = 0 ) THEN RETURN; END_IF
  // dec remaining parameter(s)
  ParameterCnt := ParameterCnt - 1;
  // Create log entry for JointPosition.J1
  CreateLogMessagePara1 ( Timestamp   := AxesGroup.State.SystemTime,
                          MessageType := MessageType.CMD,
                          Severity    := Severity.DEBUG,
                          MessageCode := 0,
                          MessageText := 'Command.JointPosition.J1 = {1}',
                          Para1       :=  REAL_TO_STRING(_command.JointPosition.J1));

  // Return if no parameter is remaining...
  IF ( ParameterCnt = 0 ) THEN RETURN; END_IF
  // dec remaining parameter(s)
  ParameterCnt := ParameterCnt - 1;
  // Create log entry for JointPosition.J2
  CreateLogMessagePara1 ( Timestamp   := AxesGroup.State.SystemTime,
                          MessageType := MessageType.CMD,
                          Severity    := Severity.DEBUG,
                          MessageCode := 0,
                          MessageText := 'Command.JointPosition.J2 = {1}',
                          Para1       :=  REAL_TO_STRING(_command.JointPosition.J2));

  // Return if no parameter is remaining...
  IF ( ParameterCnt = 0 ) THEN RETURN; END_IF
  // dec remaining parameter(s)
  ParameterCnt := ParameterCnt - 1;
  // Create log entry for JointPosition.J3
  CreateLogMessagePara1 ( Timestamp   := AxesGroup.State.SystemTime,
                          MessageType := MessageType.CMD,
                          Severity    := Severity.DEBUG,
                          MessageCode := 0,
                          MessageText := 'Command.JointPosition.J3 = {1}',
                          Para1       :=  REAL_TO_STRING(_command.JointPosition.J3));

  // Return if no parameter is remaining...
  IF ( ParameterCnt = 0 ) THEN RETURN; END_IF
  // dec remaining parameter(s)
  ParameterCnt := ParameterCnt - 1;
  // Create log entry for JointPosition.J4
  CreateLogMessagePara1 ( Timestamp   := AxesGroup.State.SystemTime,
                          MessageType := MessageType.CMD,
                          Severity    := Severity.DEBUG,
                          MessageCode := 0,
                          MessageText := 'Command.JointPosition.J4 = {1}',
                          Para1       :=  REAL_TO_STRING(_command.JointPosition.J4));

  // Return if no parameter is remaining...
  IF ( ParameterCnt = 0 ) THEN RETURN; END_IF
  // dec remaining parameter(s)
  ParameterCnt := ParameterCnt - 1;
  // Create log entry for JointPosition.J5
  CreateLogMessagePara1 ( Timestamp   := AxesGroup.State.SystemTime,
                          MessageType := MessageType.CMD,
                          Severity    := Severity.DEBUG,
                          MessageCode := 0,
                          MessageText := 'Command.JointPosition.J5 = {1}',
                          Para1       :=  REAL_TO_STRING(_command.JointPosition.J5));

  // Return if no parameter is remaining...
  IF ( ParameterCnt = 0 ) THEN RETURN; END_IF
  // dec remaining parameter(s)
  ParameterCnt := ParameterCnt - 1;
  // Create log entry for JointPosition.J6
  CreateLogMessagePara1 ( Timestamp   := AxesGroup.State.SystemTime,
                          MessageType := MessageType.CMD,
                          Severity    := Severity.DEBUG,
                          MessageCode := 0,
                          MessageText := 'Command.JointPosition.J6 = {1}',
                          Para1       :=  REAL_TO_STRING(_command.JointPosition.J6));

  // Return if no parameter is remaining...
  IF ( ParameterCnt = 0 ) THEN RETURN; END_IF
  // dec remaining parameter(s)
  ParameterCnt := ParameterCnt - 1;
  // Create log entry for JointPosition.E1
  CreateLogMessagePara1 ( Timestamp   := AxesGroup.State.SystemTime,
                          MessageType := MessageType.CMD,
                          Severity    := Severity.DEBUG,
                          MessageCode := 0,
                          MessageText := 'Command.JointPosition.E1 = {1}',
                          Para1       :=  REAL_TO_STRING(_command.JointPosition.E1));

  // Return if no parameter is remaining...
  IF ( ParameterCnt = 0 ) THEN RETURN; END_IF
  // dec remaining parameter(s)
  ParameterCnt := ParameterCnt - 1;
  // Create log entry for Manipulation
  CreateLogMessagePara1 ( Timestamp   := AxesGroup.State.SystemTime,
                          MessageType := MessageType.CMD,
                          Severity    := Severity.DEBUG,
                          MessageCode := 0,
                          MessageText := 'Command.Manipulation = {1}',
                          Para1       :=  BOOL_TO_STRING(_command.Manipulation));

  // Return if no parameter is remaining...
  IF ( ParameterCnt = 0 ) THEN RETURN; END_IF
  // dec remaining parameter(s)
  ParameterCnt := ParameterCnt - 1;
  // Create log entry for Reserve2
  CreateLogMessagePara1 ( Timestamp   := AxesGroup.State.SystemTime,
                          MessageType := MessageType.CMD,
                          Severity    := Severity.DEBUG,
                          MessageCode := 0,
                          MessageText := 'Command.Reserve2 = {1}',
                          Para1       :=  BYTE_TO_STRING(_command.Reserve2));

  // Return if no parameter is remaining...
  IF ( ParameterCnt = 0 ) THEN RETURN; END_IF
  // dec remaining parameter(s)
  ParameterCnt := ParameterCnt - 1;
  // Create log entry for MoveTime
  CreateLogMessagePara1 ( Timestamp   := AxesGroup.State.SystemTime,
                          MessageType := MessageType.CMD,
                          Severity    := Severity.DEBUG,
                          MessageCode := 0,
                          MessageText := 'Command.MoveTime = {1}',
                          Para1       :=  UINT_TO_STRING(_command.MoveTime));

  // Return if no parameter is remaining...
  IF ( ParameterCnt = 0 ) THEN RETURN; END_IF
  // dec remaining parameter(s)
  ParameterCnt := ParameterCnt - 1;
  // Create log entry for JointPosition.E2
  CreateLogMessagePara1 ( Timestamp   := AxesGroup.State.SystemTime,
                          MessageType := MessageType.CMD,
                          Severity    := Severity.DEBUG,
                          MessageCode := 0,
                          MessageText := 'Command.JointPosition.E2 = {1}',
                          Para1       :=  REAL_TO_STRING(_command.JointPosition.E2));

  // Return if no parameter is remaining...
  IF ( ParameterCnt = 0 ) THEN RETURN; END_IF
  // dec remaining parameter(s)
  ParameterCnt := ParameterCnt - 1;
  // Create log entry for JointPosition.E3
  CreateLogMessagePara1 ( Timestamp   := AxesGroup.State.SystemTime,
                          MessageType := MessageType.CMD,
                          Severity    := Severity.DEBUG,
                          MessageCode := 0,
                          MessageText := 'Command.JointPosition.E3 = {1}',
                          Para1       :=  REAL_TO_STRING(_command.JointPosition.E3));

  // Return if no parameter is remaining...
  IF ( ParameterCnt = 0 ) THEN RETURN; END_IF
  // dec remaining parameter(s)
  ParameterCnt := ParameterCnt - 1;
  // Create log entry for JointPosition.E4
  CreateLogMessagePara1 ( Timestamp   := AxesGroup.State.SystemTime,
                          MessageType := MessageType.CMD,
                          Severity    := Severity.DEBUG,
                          MessageCode := 0,
                          MessageText := 'Command.JointPosition.E4 = {1}',
                          Para1       :=  REAL_TO_STRING(_command.JointPosition.E4));

  // Return if no parameter is remaining...
  IF ( ParameterCnt = 0 ) THEN RETURN; END_IF
  // dec remaining parameter(s)
  ParameterCnt := ParameterCnt - 1;
  // Create log entry for JointPosition.E5
  CreateLogMessagePara1 ( Timestamp   := AxesGroup.State.SystemTime,
                          MessageType := MessageType.CMD,
                          Severity    := Severity.DEBUG,
                          MessageCode := 0,
                          MessageText := 'Command.JointPosition.E5 = {1}',
                          Para1       :=  REAL_TO_STRING(_command.JointPosition.E5));

  // Return if no parameter is remaining...
  IF ( ParameterCnt = 0 ) THEN RETURN; END_IF
  // dec remaining parameter(s)
  ParameterCnt := ParameterCnt - 1;
  // Create log entry for JointPosition.E6
  CreateLogMessagePara1 ( Timestamp   := AxesGroup.State.SystemTime,
                          MessageType := MessageType.CMD,
                          Severity    := Severity.DEBUG,
                          MessageCode := 0,
                          MessageText := 'Command.JointPosition.E6 = {1}',
                          Para1       :=  REAL_TO_STRING(_command.JointPosition.E6));

END_METHOD

METHOD FB_init : BOOL
VAR_INPUT
  /// if TRUE, the retain variables are initialized (warm start / cold start)
  bInitRetains : BOOL;
  /// if TRUE, the instance afterwards gets moved into the copy code (online change)
  bInCopyCode  : BOOL;
END_VAR

  MyType := 'MC_MoveAxesAbsoluteFB';

  ExecMode     := ExecutionMode.SEQUENCE_PRIMARY;
  Priority     := PriorityLevel.NORMAL;
  AbortingMode := AbortingModeEnum.BUFFER;
  SequenceFlag := SequenceFlagEnum.PRIMARY_SEQUENCE;

END_METHOD

METHOD PROTECTED OnExecRun : DINT
VAR_IN_OUT
  /// Robot assignment of function
  AxesGroup : AxesGroup;
END_VAR

  // call base implementation
  SUPER^.OnExecRun(AxesGroup := AxesGroup);

  CASE _stepCmd OF

    00:  IF ( _execute_R.Q ) AND ( NOT Error)
         THEN
           // Check function is supported and parameter are valid ?
           IF (( CheckFunctionSupported( AxesGroup := AxesGroup )) AND
               ( CheckParameterValid   ( AxesGroup := AxesGroup )))
           THEN
             // set busy flag
             Busy := TRUE;
             // Reset command outputs
             SysDepMemSet(pDest := ADR(OutCmd), Value := 0, DataLen := SIZEOF(OutCmd));
             // apply command parameter
            _parCmd := ParCmd;
             // init parameter sequence
            _command.ParSeq := 1;
             // create command data
             CommandData := CreateCommandPayload(AxesGroup := AxesGroup);
             // Add command to active command register
            _uniqueID := AxesGroup.Acyclic.ActiveCommandRegister.AddCmd( pCommandFB := ADR(THIS^ ));
             // set timeout
             SetTimeout(PT := _timeoutCmd, rTimer := _timerCmd);
             // inc step counter
            _stepCmd := _stepCmd + 1;
           END_IF
         END_IF

    01:  // Wait for responce received
         IF ( _responseReceived )
         THEN
           // reset response received flag
          _responseReceived := FALSE;
           // reset Active flag
           Active := FALSE;

           CASE  _response.State
           OF
             CmdMessageState.BUFFERED    : CommandBuffered    := TRUE;
             CmdMessageState.ACTIVE      : Active             := TRUE;
                                           // Update results
                                           OutCmd.FollowID    := _response.OriginID;
                                           OutCmd.Progress    :=  PERCENT_UINT_TO_REAL( Value := _response.Progress, IsOptional := FALSE);

             CmdMessageState.INTERRUPTED : CommandInterrupted := TRUE;
             CmdMessageState.DONE        : Done               := TRUE;
             CmdMessageState.ABORTED     : CommandAborted     := TRUE;
             CmdMessageState.ERROR       : Error              := TRUE;
           END_CASE

           // Done, Aborted or Error ?
           IF (_response.State >= CmdMessageState.DONE )
           THEN
             // Reset busy flag
             Busy := FALSE;
             // Update results
             OutCmd.FollowID          := _response.OriginID;
             OutCmd.Progress          :=  PERCENT_UINT_TO_REAL( Value := _response.Progress, IsOptional := FALSE);
             // set timeout
             SetTimeout(PT := _timeoutCmd, rTimer := _timerCmd);
             // inc step counter
            _stepCmd := _stepCmd + 1;
           END_IF
         END_IF

    02: IF ( NOT Execute)
        THEN
          Reset();
        END_IF

  ELSE
    // invalid step
    ErrorID := RobotLibraryErrorIdEnum.ERR_INVALID_STEP;
  END_CASE

  // Reset FB
  IF ( NOT Execute )
  THEN
    Reset();
  END_IF

END_METHOD

METHOD INTERNAL ParseResponsePayload : DINT
VAR_INPUT
  /// Response data
  ResponseData : RobotLibraryResponseDataFB;
  /// Timestamp
  Timestamp    : SystemTime;
END_VAR
VAR
  /// Parameter count
 _parameterCnt : DINT;
END_VAR
// Table 6-262: Received CMD payload (RC to PLC) of "MoveAxesAbsolute"
// --------------------------
// Header
// --------------------------
// Byte 00 : USINT   - ParSeq | State
// Byte 01 : SINT    - AlarmMessageSeverity
// Byte 02 : UINT    - AlarmMessageCode HB
// Byte 03 :         - AlarmMessageCode LB
// --------------------------
// Datablock
// --------------------------
// Byte 04 : USINT   - InvocationCounter
// Byte 05 : SINT    - Reserve
// Byte 06 : INT     - OriginID LW HB
// Byte 07 :         - OriginID LW LB
// Byte 08 : UINT    - Progress LW HB
// Byte 09 :         - Progress LW LB

  // call base implementation to parse the header from payload buffer
  ResponseData.PayloadPtr := SUPER^.ParseResponsePayload(ResponseData := ResponseData, Timestamp := Timestamp);

  // copy parsed header to response
  _response.ParSeq               := _rspHeader.ParSeq;
  _response.State                := _rspHeader.State;
  _response.AlarmMessageSeverity := _rspHeader.AlarmMessageSeverity;
  _response.AlarmMessageCode     := _rspHeader.AlarmMessageCode;

  // Check payload remaining ?
  IF ( ResponseData.IsPayloadRemaining)
  THEN
    // Get Response.InvocationCounter
   _response.InvocationCounter := ResponseData.GetUsint();
    // inc parameter counter
   _parameterCnt := _parameterCnt + 1;
  END_IF

  // Check payload remaining ?
  IF ( ResponseData.IsPayloadRemaining)
  THEN
    // Get Response.Reserve
   _response.Reserve := ResponseData.GetSint();
    // inc parameter counter
   _parameterCnt := _parameterCnt + 1;
  END_IF

  // Check payload remaining ?
  IF ( ResponseData.IsPayloadRemaining)
  THEN
    // Get Response.OriginID
   _response.OriginID := ResponseData.GetInt();
    // inc parameter counter
   _parameterCnt := _parameterCnt + 1;
  END_IF

  // Check payload remaining ?
  IF ( ResponseData.IsPayloadRemaining)
  THEN
    // Get Response.Progress
   _response.Progress := ResponseData.GetUint();
    // inc parameter counter
   _parameterCnt := _parameterCnt + 1;
  END_IF

  // Create logging
  ParseResponsePayloadLog(ResponseData := ResponseData, Timestamp := Timestamp, ParameterCnt := _parameterCnt);

END_METHOD

METHOD INTERNAL ParseResponsePayloadLog
VAR_INPUT
  /// Response data
  ResponseData : RobotLibraryResponseDataFB;
  /// Timestamp
  Timestamp    : SystemTime;
  /// Parameter count
  ParameterCnt : DINT;
END_VAR

  // Create log entry for Parameter start
  CreateLogMessagePara1 ( Timestamp   := Timestamp,
                          MessageType := MessageType.CMD,
                          Severity    := Severity.DEBUG,
                          MessageCode := 0,
                          MessageText := '{1} parameter(s) to parse from the response data:',
                          Para1       := DINT_TO_STRING(ParameterCnt));

  // Return if no parameter is remaining...
  IF ( ParameterCnt = 0 ) THEN RETURN; END_IF
  // dec remaining parameter(s)
  ParameterCnt := ParameterCnt - 1;
  // Create log entry for InvocationCounter
  CreateLogMessagePara1 ( Timestamp   := Timestamp,
                          MessageType := MessageType.CMD,
                          Severity    := Severity.DEBUG,
                          MessageCode := 0,
                          MessageText := 'Response.InvocationCounter = {1}',
                          Para1       :=  USINT_TO_STRING(_response.InvocationCounter));

  // Return if no parameter is remaining...
  IF ( ParameterCnt = 0 ) THEN RETURN; END_IF
  // dec remaining parameter(s)
  ParameterCnt := ParameterCnt - 1;
  // Create log entry for Reserve
  CreateLogMessagePara1 ( Timestamp   := Timestamp,
                          MessageType := MessageType.CMD,
                          Severity    := Severity.DEBUG,
                          MessageCode := 0,
                          MessageText := 'Response.Reserve = {1}',
                          Para1       :=  SINT_TO_STRING(_response.Reserve));

  // Return if no parameter is remaining...
  IF ( ParameterCnt = 0 ) THEN RETURN; END_IF
  // dec remaining parameter(s)
  ParameterCnt := ParameterCnt - 1;
  // Create log entry for OriginID
  CreateLogMessagePara1 ( Timestamp   := Timestamp,
                          MessageType := MessageType.CMD,
                          Severity    := Severity.DEBUG,
                          MessageCode := 0,
                          MessageText := 'Response.OriginID = {1}',
                          Para1       :=  INT_TO_STRING(_response.OriginID));

  // Return if no parameter is remaining...
  IF ( ParameterCnt = 0 ) THEN RETURN; END_IF
  // dec remaining parameter(s)
  ParameterCnt := ParameterCnt - 1;
  // Create log entry for Progress
  CreateLogMessagePara1 ( Timestamp   := Timestamp,
                          MessageType := MessageType.CMD,
                          Severity    := Severity.DEBUG,
                          MessageCode := 0,
                          MessageText := 'Response.Progress = {1}',
                          Para1       :=  UINT_TO_STRING(_response.Progress));

END_METHOD

METHOD PROTECTED Reset : DINT
VAR_INPUT
END_VAR

  Reset := SUPER^.Reset();

  Done               := FALSE;
  Busy               := FALSE;
  Active             := FALSE;
  CommandBuffered    := FALSE;
  CommandAborted     := FALSE;
  CommandInterrupted := FALSE;

END_METHOD
